Yaskawa INFORM job: A_ROOF_UPPER_0614_2_PL8.JBI

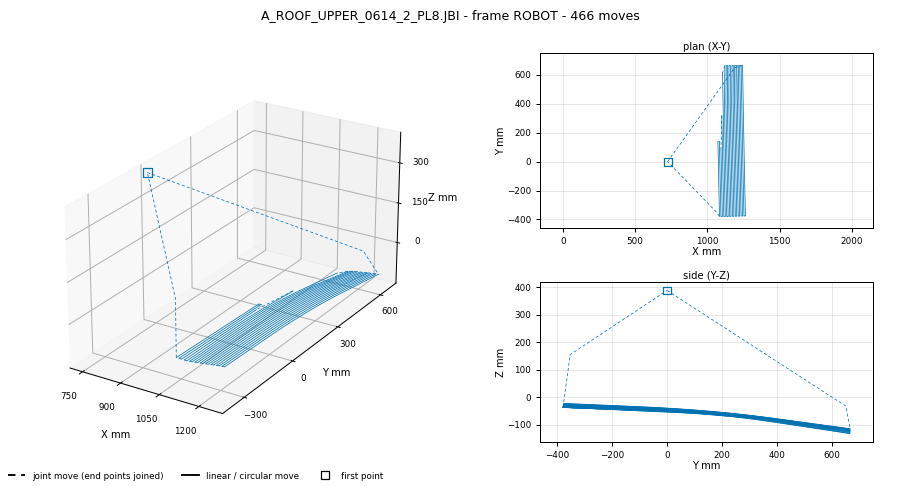
[picture p0: tool path of A_ROOF_UPPER_0614_2_PL8.JBI in frame ROBOT, 466 of 466 moves have a stored position in this frame; points joined in program order, loops and branches not executed]
/JOB
//NAME A_ROOF_UPPER_0614_2_PL8
//POS
///NPOS 466,0,0,0,0,0
///TOOL 0
///USER 0
///POSTYPE ROBOT
///RECTAN
///RCONF 1,0,0,0,0,0,0,0,0,0,0,0,0,0,0,0,0,0,0,0,0,0,0,0
C00000=725.000,0.000,388.500,-180.000,-0.000,0.000
///USER 0
///POSTYPE ROBOT
///RECTAN
C00001=1189.429,650.218,-32.227,172.053,-4.343,0.974
C00002=1243.739,665.281,-114.128,172.020,-4.282,1.414
C00003=1244.570,615.748,-107.360,172.042,-4.322,1.126
C00004=1248.336,391.180,-76.679,172.246,-4.167,0.979
C00005=1248.738,367.260,-73.517,172.471,-4.008,0.970
C00006=1249.092,346.433,-70.842,172.708,-3.888,0.966
C00007=1249.451,325.475,-68.240,172.968,-3.789,0.966
C00008=1249.796,305.508,-65.842,173.226,-3.716,0.968
C00009=1250.146,285.539,-63.530,173.487,-3.660,0.973
C00010=1250.497,265.663,-61.313,173.744,-3.621,0.979
C00011=1250.856,245.682,-59.173,174.000,-3.596,0.988
C00012=1251.235,224.702,-57.018,174.263,-3.583,0.998
C00013=1251.619,203.718,-54.952,174.521,-3.582,1.010
C00014=1252.006,182.729,-52.977,174.773,-3.593,1.023
C00015=1252.415,160.820,-51.011,175.027,-3.617,1.037
C00016=1252.831,138.821,-49.128,175.274,-3.653,1.053
C00017=1253.250,116.819,-47.334,175.514,-3.702,1.070
C00018=1253.692,93.813,-45.555,175.757,-3.765,1.088
C00019=1254.138,70.801,-43.865,175.991,-3.840,1.107
C00020=1254.589,47.783,-42.265,176.219,-3.924,1.127
C00021=1255.064,23.760,-40.691,176.449,-4.023,1.148
C00022=1255.542,-0.269,-39.207,176.673,-4.129,1.169
C00023=1256.026,-24.305,-37.813,176.890,-4.242,1.190
C00024=1256.533,-49.345,-36.455,177.109,-4.364,1.211
C00025=1257.044,-74.393,-35.191,177.323,-4.490,1.232
C00026=1257.558,-99.363,-34.023,177.531,-4.617,1.253
C00027=1262.246,-325.192,-24.300,177.735,-4.744,1.362
C00028=1263.282,-375.135,-22.149,177.733,-4.743,1.386
C00029=1253.337,-375.387,-23.203,177.732,-4.743,1.394
C00030=1252.299,-325.442,-25.310,177.735,-4.744,1.363
C00031=1247.595,-99.606,-34.838,177.531,-4.617,1.253
C00032=1247.079,-74.637,-35.984,177.323,-4.490,1.233
C00033=1246.565,-49.589,-37.227,177.109,-4.364,1.211
C00034=1246.057,-24.549,-38.563,176.890,-4.242,1.190
C00035=1245.572,-0.513,-39.937,176.673,-4.129,1.169
C00036=1245.092,23.516,-41.404,176.449,-4.023,1.148
C00037=1244.616,47.539,-42.961,176.219,-3.924,1.127
C00038=1244.165,70.557,-44.547,175.991,-3.840,1.107
C00039=1243.718,93.569,-46.224,175.757,-3.765,1.088
C00040=1243.275,116.575,-47.994,175.514,-3.702,1.070
C00041=1242.855,138.578,-49.780,175.274,-3.653,1.053
C00042=1242.439,160.575,-51.657,175.027,-3.617,1.037
C00043=1242.030,182.485,-53.620,174.773,-3.593,1.022
C00044=1241.642,203.473,-55.593,174.521,-3.582,1.009
C00045=1241.259,224.457,-57.659,174.263,-3.583,0.997
C00046=1240.879,245.434,-59.817,174.000,-3.596,0.986
C00047=1240.523,265.414,-61.962,173.744,-3.621,0.978
C00048=1240.171,285.288,-64.184,173.487,-3.660,0.971
C00049=1239.822,305.255,-66.507,173.226,-3.716,0.966
C00050=1239.477,325.219,-68.917,172.968,-3.789,0.964
C00051=1239.119,346.174,-71.538,172.709,-3.888,0.964
C00052=1238.768,366.999,-74.233,172.472,-4.008,0.968
C00053=1238.368,390.913,-77.423,172.246,-4.167,0.975
C00054=1234.646,615.465,-108.292,172.043,-4.324,1.109
C00055=1233.823,664.993,-115.099,172.011,-4.264,1.539
C00056=1223.907,664.704,-116.071,172.022,-4.285,1.389
C00057=1224.720,615.181,-109.222,172.045,-4.328,1.079
C00058=1228.400,390.647,-78.167,172.246,-4.168,0.972
C00059=1228.796,366.737,-74.949,172.472,-4.009,0.965
C00060=1229.147,345.916,-72.234,172.709,-3.889,0.962
C00061=1229.504,324.965,-69.594,172.968,-3.790,0.962
C00062=1229.847,305.004,-67.172,173.227,-3.716,0.964
C00063=1230.195,285.038,-64.840,173.487,-3.661,0.969
C00064=1230.546,265.166,-62.611,173.745,-3.622,0.976
C00065=1230.903,245.187,-60.461,174.000,-3.596,0.985
C00066=1231.282,224.210,-58.299,174.263,-3.583,0.996
C00067=1231.666,203.228,-56.234,174.521,-3.582,1.008
C00068=1232.054,182.240,-54.262,174.773,-3.593,1.021
C00069=1232.463,160.332,-52.302,175.027,-3.617,1.036
C00070=1232.880,138.334,-50.431,175.275,-3.653,1.052
C00071=1233.299,116.331,-48.654,175.514,-3.703,1.069
C00072=1233.743,93.326,-46.894,175.757,-3.765,1.088
C00073=1234.191,70.313,-45.228,175.991,-3.840,1.107
C00074=1234.644,47.295,-43.657,176.219,-3.924,1.127
C00075=1235.121,23.272,-42.115,176.449,-4.023,1.148
C00076=1235.601,-0.756,-40.668,176.673,-4.129,1.169
C00077=1236.087,-24.792,-39.313,176.890,-4.242,1.190
C00078=1236.598,-49.832,-37.998,177.109,-4.364,1.211
C00079=1237.113,-74.880,-36.777,177.323,-4.490,1.233
C00080=1237.630,-99.850,-35.654,177.531,-4.617,1.253
C00081=1242.351,-325.692,-26.320,177.734,-4.744,1.364
C00082=1243.394,-375.638,-24.255,177.733,-4.743,1.386
C00083=1233.450,-375.899,-25.309,177.782,-4.867,1.385
C00084=1232.404,-325.951,-27.330,177.783,-4.867,1.369
C00085=1227.667,-100.100,-36.468,177.580,-4.745,1.262
C00086=1227.148,-75.130,-37.570,177.372,-4.623,1.242
C00087=1226.631,-50.081,-38.769,177.158,-4.501,1.221
C00088=1226.118,-25.039,-40.063,176.937,-4.382,1.200
C00089=1225.631,-1.002,-41.397,176.718,-4.273,1.180
C00090=1225.149,23.028,-42.827,176.492,-4.172,1.159
C00091=1224.691,46.055,-44.287,176.267,-4.082,1.140
C00092=1224.236,69.074,-45.840,176.036,-4.001,1.121
C00093=1223.787,92.088,-47.487,175.796,-3.931,1.102
C00094=1223.362,114.097,-49.155,175.560,-3.875,1.085
C00095=1222.940,136.101,-50.915,175.316,-3.831,1.069
C00096=1222.525,158.020,-52.764,175.065,-3.798,1.053
C00097=1222.133,179.014,-54.627,174.817,-3.780,1.040
C00098=1221.744,200.003,-56.583,174.561,-3.772,1.027
C00099=1221.360,220.986,-58.635,174.297,-3.778,1.016
C00100=1220.997,240.970,-60.681,174.042,-3.795,1.006
C00101=1220.642,260.854,-62.807,173.783,-3.823,0.998
C00102=1220.289,280.824,-65.035,173.517,-3.865,0.991
C00103=1219.941,300.791,-67.357,173.248,-3.923,0.987
C00104=1219.596,320.754,-69.774,172.980,-3.998,0.984
C00105=1219.259,340.595,-72.269,172.721,-4.092,0.984
C00106=1218.907,361.536,-74.999,172.465,-4.215,0.988
C00107=1218.527,384.455,-78.089,172.229,-4.375,0.996
C00108=1217.998,417.090,-82.628,171.990,-4.603,1.009
C00109=1214.953,615.116,-110.490,171.985,-4.594,1.073
C00110=1214.190,664.623,-117.456,171.968,-4.565,1.281
C00111=1204.182,664.600,-118.494,171.912,-4.846,1.173
C00112=1204.954,615.099,-111.491,171.922,-4.863,1.056
C00113=1208.251,403.160,-81.508,172.008,-4.769,1.030
C00114=1208.674,377.272,-77.910,172.222,-4.570,1.018
C00115=1209.020,356.332,-75.085,172.461,-4.421,1.011
C00116=1209.355,336.382,-72.485,172.722,-4.302,1.007
C00117=1209.692,316.541,-69.991,172.994,-4.207,1.007
C00118=1210.019,297.569,-67.698,173.257,-4.134,1.009
C00119=1210.368,277.602,-65.380,173.534,-4.072,1.013
C00120=1210.721,257.629,-63.159,173.806,-4.026,1.019
C00121=1211.077,237.745,-61.042,174.070,-3.993,1.027
C00122=1211.440,217.760,-59.007,174.331,-3.972,1.035
C00123=1211.806,197.771,-57.062,174.586,-3.962,1.046
C00124=1212.195,176.781,-55.116,174.847,-3.965,1.057
C00125=1212.589,155.786,-53.265,175.100,-3.979,1.070
C00126=1212.985,134.863,-51.512,175.345,-4.006,1.084
C00127=1213.407,112.858,-49.764,175.594,-4.045,1.100
C00128=1213.834,90.847,-48.109,175.835,-4.097,1.116
C00129=1214.265,68.830,-46.548,176.068,-4.159,1.133
C00130=1214.720,45.809,-45.009,176.304,-4.235,1.152
C00131=1215.179,22.782,-43.565,176.532,-4.321,1.171
C00132=1215.663,-1.249,-42.153,176.761,-4.418,1.190
C00133=1216.152,-25.287,-40.836,176.983,-4.522,1.210
C00134=1216.665,-50.331,-39.564,177.205,-4.636,1.231
C00135=1217.184,-75.381,-38.386,177.421,-4.753,1.251
C00136=1217.705,-100.353,-37.305,177.628,-4.871,1.270
C00137=1222.459,-326.211,-28.354,177.830,-4.989,1.374
C00138=1223.509,-376.162,-26.375,177.829,-4.988,1.386
C00139=1213.569,-376.423,-27.454,177.874,-5.109,1.389
C00140=1212.515,-326.472,-29.394,177.875,-5.109,1.379
C00141=1207.745,-100.606,-38.163,177.674,-4.996,1.279
C00142=1207.223,-75.634,-39.224,177.467,-4.883,1.260
C00143=1206.702,-50.583,-40.382,177.251,-4.771,1.240
C00144=1206.187,-25.538,-41.635,177.027,-4.662,1.220
C00145=1205.697,-1.499,-42.934,176.803,-4.562,1.201
C00146=1205.211,22.535,-44.329,176.570,-4.469,1.182
C00147=1204.751,45.563,-45.759,176.339,-4.389,1.164
C00148=1204.295,68.585,-47.284,176.099,-4.318,1.146
C00149=1203.863,90.602,-48.835,175.861,-4.260,1.130
C00150=1203.436,112.614,-50.480,175.615,-4.214,1.114
C00151=1203.033,133.622,-52.140,175.372,-4.180,1.100
C00152=1202.635,154.546,-53.884,175.122,-4.159,1.087
C00153=1202.241,175.542,-55.729,174.864,-4.149,1.074
C00154=1201.870,195.536,-57.576,174.610,-4.151,1.064
C00155=1201.503,215.526,-59.512,174.349,-4.166,1.055
C00156=1201.143,235.421,-61.533,174.085,-4.191,1.046
C00157=1200.784,255.397,-63.656,173.813,-4.230,1.040
C00158=1200.449,274.376,-65.763,173.549,-4.279,1.035
C00159=1200.118,293.351,-67.959,173.279,-4.341,1.032
C00160=1199.793,312.213,-70.232,173.009,-4.416,1.030
C00161=1199.471,331.175,-72.609,172.739,-4.507,1.030
C00162=1199.153,350.136,-75.076,172.477,-4.618,1.033
C00163=1198.823,370.087,-77.763,172.221,-4.761,1.040
C00164=1198.434,393.997,-81.090,171.994,-4.957,1.052
C00165=1198.074,417.105,-84.377,171.858,-5.130,1.063
C00166=1198.550,615.125,-112.440,171.859,-5.131,1.053
C00167=1198.667,664.630,-119.456,171.852,-5.120,1.130
C00168=1189.050,664.613,-120.644,171.795,-5.403,1.029
C00169=1188.865,615.115,-113.579,171.795,-5.403,1.027
C00170=1188.115,416.320,-85.209,171.793,-5.389,1.090
C00171=1188.557,388.647,-81.242,171.950,-5.168,1.076
C00172=1188.910,366.863,-78.195,172.180,-4.979,1.064
C00173=1189.221,347.902,-75.628,172.441,-4.841,1.057
C00174=1189.538,328.941,-73.152,172.717,-4.729,1.054
C00175=1189.860,309.978,-70.769,172.996,-4.635,1.053
C00176=1190.184,291.118,-68.492,173.272,-4.556,1.054
C00177=1190.515,272.142,-66.294,173.548,-4.489,1.056
C00178=1190.851,253.162,-64.188,173.818,-4.433,1.060
C00179=1191.209,233.186,-62.068,174.096,-4.389,1.066
C00180=1191.569,213.291,-60.053,174.367,-4.359,1.074
C00181=1191.936,193.300,-58.122,174.632,-4.340,1.082
C00182=1192.308,173.305,-56.284,174.891,-4.334,1.092
C00183=1192.703,152.308,-54.451,175.154,-4.339,1.104
C00184=1193.103,131.306,-52.712,175.410,-4.356,1.116
C00185=1193.505,110.373,-51.073,175.656,-4.386,1.130
C00186=1193.933,88.361,-49.445,175.906,-4.429,1.145
C00187=1194.366,66.342,-47.912,176.149,-4.482,1.160
C00188=1194.804,44.317,-46.471,176.382,-4.546,1.177
C00189=1195.266,21.288,-45.059,176.617,-4.622,1.194
C00190=1195.732,-1.749,-43.739,176.843,-4.707,1.212
C00191=1196.224,-25.789,-42.458,177.069,-4.801,1.230
C00192=1196.720,-49.837,-41.271,177.286,-4.902,1.249
C00193=1197.240,-74.806,-40.133,177.502,-5.009,1.268
C00194=1197.787,-100.862,-39.044,177.719,-5.121,1.287
C00195=1202.573,-326.734,-30.447,177.917,-5.229,1.384
C00196=1203.630,-376.687,-28.546,177.916,-5.228,1.394
C00197=1193.692,-376.950,-29.649,177.957,-5.346,1.400
C00198=1192.632,-326.997,-31.513,177.958,-5.347,1.390
C00199=1187.832,-101.118,-39.946,177.760,-5.245,1.295
C00200=1187.282,-75.061,-41.016,177.544,-5.138,1.276
C00201=1186.761,-50.091,-42.135,177.328,-5.036,1.258
C00202=1186.263,-26.043,-43.305,177.109,-4.941,1.240
C00203=1185.770,-2.000,-44.570,176.880,-4.851,1.222
C00204=1185.302,21.036,-45.876,176.651,-4.772,1.205
C00205=1184.839,44.067,-47.274,176.412,-4.701,1.189
C00206=1184.401,66.092,-48.705,176.175,-4.641,1.173
C00207=1183.967,88.111,-50.228,175.928,-4.593,1.158
C00208=1183.558,109.128,-51.774,175.684,-4.556,1.144
C00209=1183.154,130.061,-53.404,175.433,-4.531,1.132
C00210=1182.755,151.064,-55.134,175.172,-4.518,1.120
C00211=1182.378,171.066,-56.872,174.916,-4.517,1.110
C00212=1182.005,191.061,-58.703,174.652,-4.528,1.100
C00213=1181.638,211.053,-60.627,174.382,-4.551,1.092
C00214=1181.277,230.948,-62.638,174.105,-4.587,1.086
C00215=1180.937,249.931,-64.649,173.835,-4.633,1.081
C00216=1180.602,268.912,-66.750,173.559,-4.693,1.078
C00217=1180.273,287.783,-68.933,173.280,-4.765,1.076
C00218=1179.947,306.749,-71.221,172.995,-4.849,1.076
C00219=1179.626,325.713,-73.605,172.709,-4.946,1.077
C00220=1179.310,344.675,-76.086,172.422,-5.059,1.081
C00221=1179.002,363.500,-78.644,172.142,-5.195,1.087
C00222=1178.681,383.439,-81.448,171.901,-5.376,1.099
C00223=1178.163,416.202,-86.182,171.725,-5.655,1.118
C00224=1179.134,615.111,-114.770,171.734,-5.679,1.000
C00225=1179.376,664.602,-121.883,171.741,-5.689,0.926
C00226=1170.628,664.605,-123.074,171.686,-5.975,0.835
C00227=1170.148,615.119,-115.932,171.671,-5.954,0.981
C00228=1168.215,416.580,-87.274,171.655,-5.926,1.146
C00229=1168.414,403.116,-85.300,171.691,-5.823,1.140
C00230=1168.838,376.249,-81.401,171.878,-5.557,1.120
C00231=1169.127,358.289,-78.872,172.140,-5.399,1.110
C00232=1169.418,340.455,-76.449,172.419,-5.274,1.104
C00233=1169.717,322.482,-74.096,172.700,-5.164,1.101
C00234=1170.020,304.510,-71.832,172.979,-5.068,1.099
C00235=1170.346,285.544,-69.539,173.269,-4.978,1.098
C00236=1170.674,266.673,-67.354,173.554,-4.901,1.099
C00237=1171.009,247.692,-65.252,173.836,-4.835,1.101
C00238=1171.348,228.709,-63.243,174.112,-4.784,1.106
C00239=1171.693,209.721,-61.325,174.381,-4.745,1.111
C00240=1172.059,189.817,-59.410,174.657,-4.717,1.118
C00241=1172.431,169.819,-57.583,174.926,-4.701,1.127
C00242=1172.808,149.818,-55.849,175.188,-4.697,1.136
C00243=1173.189,129.811,-54.204,175.442,-4.705,1.147
C00244=1173.593,108.878,-52.579,175.698,-4.725,1.159
C00245=1174.003,87.862,-51.040,175.948,-4.757,1.172
C00246=1174.437,65.841,-49.525,176.199,-4.801,1.186
C00247=1174.876,43.815,-48.104,176.441,-4.855,1.201
C00248=1175.340,20.784,-46.718,176.683,-4.921,1.217
C00249=1175.810,-2.254,-45.427,176.915,-4.996,1.233
C00250=1176.304,-26.298,-44.177,177.146,-5.081,1.250
C00251=1176.803,-50.347,-43.023,177.367,-5.171,1.267
C00252=1177.327,-75.317,-41.921,177.585,-5.267,1.285
C00253=1177.877,-101.376,-40.869,177.800,-5.367,1.302
C00254=1182.692,-327.261,-32.593,177.997,-5.464,1.395
C00255=1183.756,-377.215,-30.762,177.996,-5.464,1.407
C00256=1173.821,-377.482,-31.885,178.031,-5.581,1.415
C00257=1172.755,-327.525,-33.683,178.033,-5.581,1.401
C00258=1167.926,-101.635,-41.814,177.838,-5.490,1.310
C00259=1167.372,-75.576,-42.848,177.622,-5.395,1.293
C00260=1166.847,-50.605,-43.934,177.404,-5.305,1.276
C00261=1166.347,-26.554,-45.073,177.182,-5.221,1.260
C00262=1165.871,-3.508,-46.255,176.958,-5.145,1.244
C00263=1165.401,19.531,-47.529,176.724,-5.075,1.229
C00264=1164.956,41.565,-48.839,176.489,-5.015,1.214
C00265=1164.515,63.594,-50.241,176.243,-4.965,1.200
C00266=1164.099,84.617,-51.669,176.000,-4.926,1.187
C00267=1163.690,105.558,-53.184,175.747,-4.897,1.175
C00268=1163.284,126.569,-54.798,175.485,-4.880,1.163
C00269=1162.902,146.577,-56.427,175.228,-4.875,1.153
C00270=1162.524,166.580,-58.148,174.961,-4.882,1.144
C00271=1162.152,186.577,-59.964,174.687,-4.902,1.136
C00272=1161.803,205.488,-61.772,174.421,-4.932,1.130
C00273=1161.459,224.477,-63.678,174.146,-4.975,1.126
C00274=1161.119,243.462,-65.675,173.865,-5.030,1.122
C00275=1160.784,262.444,-67.770,173.576,-5.099,1.120
C00276=1160.455,281.316,-69.947,173.286,-5.180,1.120
C00277=1160.147,299.292,-72.114,173.005,-5.269,1.121
C00278=1159.843,317.267,-74.370,172.722,-5.369,1.124
C00279=1159.547,335.113,-76.700,172.436,-5.482,1.128
C00280=1159.254,353.076,-79.137,172.145,-5.609,1.134
C00281=1158.982,370.049,-81.526,171.867,-5.747,1.142
C00282=1158.672,389.838,-84.407,171.642,-5.956,1.158
C00283=1158.272,415.709,-88.232,171.585,-6.187,1.174
C00284=1159.271,615.118,-117.349,171.606,-6.230,0.958
C00285=1159.517,664.594,-124.574,171.633,-6.267,0.706
C00286=1149.612,664.593,-126.030,171.572,-6.554,0.588
C00287=1149.358,615.127,-118.743,171.531,-6.500,0.952
C00288=1148.334,415.437,-89.323,171.506,-6.448,1.202
C00289=1148.805,384.623,-84.721,171.566,-6.150,1.180
C00290=1149.083,366.815,-82.112,171.830,-5.974,1.167
C00291=1149.353,349.841,-79.714,172.120,-5.836,1.159
C00292=1149.644,331.877,-77.270,172.418,-5.703,1.152
C00293=1149.941,314.032,-74.935,172.710,-5.583,1.147
C00294=1150.243,296.056,-72.677,173.000,-5.477,1.143
C00295=1150.550,278.079,-70.510,173.287,-5.384,1.141
C00296=1150.862,260.101,-68.434,173.570,-5.303,1.141
C00297=1151.195,241.218,-66.349,173.862,-5.230,1.142
C00298=1151.535,222.233,-64.351,174.150,-5.170,1.145
C00299=1151.880,203.243,-62.447,174.430,-5.122,1.149
C00300=1152.228,184.332,-60.644,174.702,-5.087,1.154
C00301=1152.582,165.330,-58.922,174.969,-5.064,1.161
C00302=1152.960,145.327,-57.205,175.240,-5.053,1.169
C00303=1153.342,125.319,-55.581,175.504,-5.054,1.178
C00304=1153.730,105.304,-54.049,175.758,-5.066,1.189
C00305=1154.140,84.363,-52.539,176.015,-5.090,1.200
C00306=1154.557,63.338,-51.116,176.264,-5.125,1.213
C00307=1154.998,41.310,-49.724,176.513,-5.170,1.226
C00308=1155.444,19.275,-48.424,176.751,-5.225,1.240
C00309=1155.915,-3.765,-47.162,176.989,-5.290,1.255
C00310=1156.392,-26.812,-45.994,177.215,-5.361,1.270
C00311=1156.895,-50.864,-44.869,177.439,-5.439,1.285
C00312=1157.421,-75.835,-43.798,177.658,-5.524,1.301
C00313=1157.975,-101.896,-42.781,177.872,-5.612,1.318
C00314=1162.819,-327.791,-34.786,178.067,-5.697,1.406
C00315=1163.889,-377.749,-33.019,178.065,-5.696,1.424
C00316=1153.956,-378.015,-34.144,178.095,-5.810,1.435
C00317=1152.884,-328.057,-35.887,178.098,-5.811,1.410
C00318=1148.006,-101.159,-43.805,177.897,-5.731,1.324
C00319=1147.450,-75.098,-44.811,177.682,-5.649,1.309
C00320=1146.921,-50.041,-45.875,177.461,-5.570,1.294
C00321=1146.419,-26.072,-46.986,177.237,-5.497,1.279
C00322=1145.942,-3.026,-48.147,177.008,-5.432,1.265
C00323=1145.469,20.015,-49.402,176.766,-5.373,1.251
C00324=1145.022,42.051,-50.697,176.524,-5.324,1.237
C00325=1144.600,63.082,-52.021,176.282,-5.284,1.225
C00326=1144.183,84.106,-53.437,176.029,-5.255,1.214
C00327=1143.772,105.048,-54.942,175.767,-5.235,1.203
C00328=1143.384,125.062,-56.474,175.507,-5.228,1.193
C00329=1143.002,145.072,-58.097,175.237,-5.231,1.185
C00330=1142.643,164.078,-59.729,174.973,-5.247,1.178
C00331=1142.291,182.997,-61.442,174.702,-5.274,1.172
C00332=1141.941,201.991,-63.254,174.423,-5.314,1.167
C00333=1141.597,220.981,-65.161,174.135,-5.367,1.164
C00334=1141.275,238.973,-67.058,173.857,-5.429,1.162
C00335=1140.961,256.861,-69.032,173.575,-5.502,1.162
C00336=1140.649,274.841,-71.107,173.287,-5.586,1.163
C00337=1140.342,292.818,-73.275,172.993,-5.683,1.165
C00338=1140.042,310.675,-75.522,172.698,-5.793,1.169
C00339=1139.746,328.640,-77.877,172.397,-5.918,1.175
C00340=1139.471,345.614,-80.191,172.109,-6.051,1.183
C00341=1139.204,362.445,-82.572,171.817,-6.197,1.192
C00342=1138.941,379.408,-85.062,171.524,-6.352,1.203
C00343=1138.535,406.032,-89.076,171.344,-8.117,1.401
C00344=1138.400,415.917,-90.582,171.339,-8.283,1.418
C00345=1140.286,615.128,-120.237,171.373,-8.347,1.185
C00346=1140.753,664.582,-127.599,171.441,-8.417,0.720
C00347=1130.859,664.438,-129.965,171.213,-8.393,0.854
C00348=1130.391,615.012,-122.427,171.167,-8.345,1.167
C00349=1128.495,415.610,-92.013,171.142,-8.273,1.414
C00350=1128.845,391.183,-88.242,171.323,-7.974,1.385
C00351=1129.105,373.942,-85.634,171.528,-7.922,1.384
C00352=1129.376,356.411,-83.063,171.815,-7.904,1.386
C00353=1129.653,338.867,-80.585,172.115,-7.878,1.388
C00354=1129.947,320.597,-78.099,172.413,-7.846,1.388
C00355=1130.252,302.036,-75.673,172.713,-7.808,1.389
C00356=1130.562,283.463,-73.344,173.011,-7.768,1.388
C00357=1130.874,265.152,-71.147,173.304,-7.719,1.387
C00358=1131.196,246.555,-69.011,173.627,-7.662,1.385
C00359=1131.523,227.947,-66.969,173.903,-7.594,1.382
C00360=1131.869,208.607,-64.955,174.185,-7.493,1.377
C00361=1132.170,191.968,-63.300,174.454,-7.420,1.373
C00362=1132.512,173.331,-61.532,174.728,-7.324,1.368
C00363=1132.862,154.589,-59.848,175.016,-7.210,1.362
C00364=1133.257,133.814,-58.115,175.384,-5.404,1.205
C00365=1133.643,113.801,-56.544,175.655,-5.402,1.213
C00366=1134.042,93.323,-55.032,175.921,-5.412,1.222
C00367=1134.248,82.850,-54.296,176.052,-5.420,1.228
C00368=1134.666,61.825,-52.889,176.309,-5.446,1.239
C00369=1135.089,40.793,-51.575,176.555,-5.481,1.250
C00370=1135.536,18.757,-50.293,176.801,-5.525,1.262
C00371=1135.990,-3.285,-49.104,177.034,-5.577,1.275
C00372=1136.469,-26.333,-47.954,177.265,-5.637,1.289
C00373=1136.972,-50.303,-46.855,177.491,-5.704,1.303
C00374=1137.502,-75.360,-45.806,177.713,-5.776,1.317
C00375=1138.059,-101.422,-44.812,177.927,-5.852,1.332
C00376=1142.950,-328.325,-37.013,178.126,-5.926,1.414
C00377=1144.025,-378.284,-35.295,178.124,-5.926,1.433
C00378=1134.095,-378.553,-36.456,178.150,-6.040,1.432
C00379=1133.018,-328.593,-38.149,178.152,-6.040,1.418
C00380=1128.115,-101.686,-45.842,177.954,-5.973,1.339
C00381=1127.556,-75.574,-46.823,177.830,-4.400,1.222
C00382=1127.123,-55.297,-47.638,177.588,-4.743,1.236
C00383=1126.707,-35.594,-48.505,177.359,-5.057,1.250
C00384=1126.239,-13.173,-49.585,177.121,-5.392,1.265
C00385=1125.797,8.243,-50.711,176.879,-5.700,1.280
C00386=1125.396,27.932,-51.829,176.632,-5.969,1.293
C00387=1125.000,47.615,-53.031,176.381,-6.207,1.306
C00388=1124.594,68.013,-54.370,176.119,-6.433,1.318
C00389=1124.188,88.681,-55.821,175.864,-6.653,1.330
C00390=1123.812,108.068,-57.270,175.585,-6.839,1.340
C00391=1123.435,127.723,-58.838,175.314,-6.996,1.349
C00392=1123.050,148.089,-60.555,175.049,-7.159,1.359
C00393=1122.703,166.733,-62.219,174.762,-7.283,1.365
C00394=1122.347,186.083,-64.041,174.481,-7.389,1.371
C00395=1122.010,204.709,-65.886,174.200,-7.477,1.375
C00396=1121.678,223.325,-67.823,173.932,-7.569,1.380
C00397=1121.373,240.656,-69.712,173.650,-7.637,1.383
C00398=1121.062,258.691,-71.764,173.384,-7.699,1.385
C00399=1120.753,276.844,-73.918,173.095,-7.752,1.387
C00400=1120.446,295.136,-76.185,172.799,-7.793,1.387
C00401=1120.141,313.696,-78.581,172.502,-7.831,1.387
C00402=1119.840,332.242,-81.075,172.202,-7.866,1.386
C00403=1119.552,350.495,-83.626,171.904,-7.897,1.385
C00404=1119.281,368.026,-86.170,171.606,-7.915,1.383
C00405=1119.016,385.542,-88.803,171.332,-7.947,1.381
C00406=1118.801,400.084,-91.046,171.151,-8.043,1.388
C00407=1118.619,412.643,-93.022,170.986,-8.214,1.405
C00408=1118.593,415.606,-93.491,170.946,-8.268,1.410
C00409=1120.778,614.897,-124.574,170.959,-8.342,1.162
C00410=1121.318,664.296,-132.280,170.991,-8.376,0.944
C00411=1105.570,614.010,-123.215,171.652,-7.951,1.120
C00412=1106.334,564.532,-116.047,171.635,-7.933,1.243
C00413=1109.667,348.539,-84.757,171.918,-7.893,1.384
C00414=1109.959,330.009,-82.171,172.217,-7.862,1.385
C00415=1110.258,311.466,-79.683,172.515,-7.826,1.386
C00416=1110.558,293.195,-77.327,172.806,-7.788,1.386
C00417=1110.869,274.627,-75.028,173.100,-7.744,1.385
C00418=1111.184,256.046,-72.825,173.386,-7.688,1.384
C00419=1111.501,237.740,-70.744,173.655,-7.626,1.382
C00420=1111.809,220.132,-68.825,173.923,-7.549,1.378
C00421=1112.123,202.516,-66.989,174.194,-7.467,1.374
C00422=1112.471,183.184,-65.070,174.471,-7.373,1.369
C00423=1112.831,163.560,-63.216,174.744,-7.262,1.364
C00424=1113.172,145.205,-61.569,175.010,-7.132,1.356
C00425=1113.560,124.566,-59.813,175.275,-6.967,1.347
C00426=1113.915,105.914,-58.310,175.527,-6.816,1.338
C00427=1114.289,86.537,-56.838,175.783,-6.625,1.327
C00428=1114.693,65.877,-55.358,176.035,-6.405,1.315
C00429=1115.096,45.490,-53.989,176.289,-6.176,1.303
C00430=1115.509,24.816,-52.692,176.538,-5.921,1.290
C00431=1115.942,3.417,-51.441,176.785,-5.622,1.275
C00432=1116.365,-17.269,-50.320,177.021,-5.324,1.261
C00433=1116.829,-39.679,-49.199,177.262,-4.988,1.246
C00434=1117.318,-63.093,-48.127,177.504,-4.605,1.229
C00435=1117.778,-84.792,-47.225,177.742,-4.223,1.214
C00436=1118.299,-109.216,-46.306,177.963,-3.788,1.198
C00437=1123.026,-328.488,-38.851,178.153,-3.420,1.301
C00438=1124.102,-378.447,-37.152,178.152,-3.419,1.324
C00439=1114.039,-378.200,-37.108,177.952,-3.411,1.315
C00440=1112.977,-328.245,-38.938,177.953,-3.412,1.297
C00441=1108.496,-117.713,-46.648,177.858,-3.621,1.191
C00442=1108.001,-94.298,-47.571,177.645,-4.042,1.206
C00443=1107.511,-70.887,-48.581,177.420,-4.461,1.222
C00444=1107.040,-48.199,-49.653,177.190,-4.840,1.238
C00445=1106.600,-26.797,-50.745,176.973,-5.170,1.253
C00446=1106.160,-5.118,-51.939,176.736,-5.491,1.267
C00447=1105.729,16.272,-53.205,176.497,-5.798,1.283
C00448=1105.304,37.655,-54.560,176.261,-6.076,1.297
C00449=1104.898,58.318,-55.956,176.017,-6.316,1.310
C00450=1104.501,78.690,-57.421,175.764,-6.536,1.322
C00451=1104.105,99.339,-58.995,175.519,-6.750,1.334
C00452=1099.944,318.457,-76.674,175.270,-6.926,1.284
C00453=1094.176,89.157,-55.681,177.767,-3.412,1.051
C00454=1102.917,-327.991,-38.766,177.753,-3.402,1.292
C00455=1103.962,-377.939,-36.741,177.752,-3.402,1.308
C00456=1093.939,-378.145,-36.643,177.752,-3.402,1.301
C00457=1092.902,-328.203,-38.807,177.753,-3.403,1.287
C00458=1084.234,88.899,-56.878,177.616,-3.744,1.079
C00459=1083.195,138.841,-59.042,177.617,-3.745,1.050
C00460=1073.262,138.575,-60.377,177.617,-3.745,1.049
C00461=1074.292,88.639,-58.075,177.616,-3.744,1.078
C00462=1082.888,-328.413,-38.847,177.753,-3.403,1.282
C00463=1083.916,-378.349,-36.545,177.752,-3.402,1.294
C00464=1066.114,-352.262,155.451,177.759,-3.407,1.176
///USER 0
///POSTYPE ROBOT
///RECTAN
C00465=725.000,0.000,388.500,-180.000,-0.000,0.000
//INST
///DATE 2021/06/15 16:23
///ATTR SC,RW,RJ
////FRAME ROBOT
///GROUP1 RB1
NOP
MOVJ C00000 VJ=100.00 PL=0
'Path Start: Op_ID_1
MOVJ C00001 VJ=25.00 PL=0
MOVJ C00002 VJ=25.00 PL=0
MOVL C00003 V=800.0 PL=8
SPYON
MOVL C00004 V=800.0 PL=8
MOVL C00005 V=800.0 PL=8
MOVL C00006 V=800.0 PL=8
MOVL C00007 V=800.0 PL=8
MOVL C00008 V=800.0 PL=8
MOVL C00009 V=800.0 PL=8
MOVL C00010 V=800.0 PL=8
MOVL C00011 V=800.0 PL=8
MOVL C00012 V=800.0 PL=8
MOVL C00013 V=800.0 PL=8
MOVL C00014 V=800.0 PL=8
MOVL C00015 V=800.0 PL=8
MOVL C00016 V=800.0 PL=8
MOVL C00017 V=800.0 PL=8
MOVL C00018 V=800.0 PL=8
MOVL C00019 V=800.0 PL=8
MOVL C00020 V=800.0 PL=8
MOVL C00021 V=800.0 PL=8
MOVL C00022 V=800.0 PL=8
MOVL C00023 V=800.0 PL=8
MOVL C00024 V=800.0 PL=8
MOVL C00025 V=800.0 PL=8
MOVL C00026 V=800.0 PL=8
MOVL C00027 V=800.0 PL=8
SPYOF
MOVL C00028 V=800.0 PL=0
MOVJ C00029 VJ=25.00 PL=0
MOVL C00030 V=800.0 PL=8
SPYON
MOVL C00031 V=800.0 PL=8
MOVL C00032 V=800.0 PL=8
MOVL C00033 V=800.0 PL=8
MOVL C00034 V=800.0 PL=8
MOVL C00035 V=800.0 PL=8
MOVL C00036 V=800.0 PL=8
MOVL C00037 V=800.0 PL=8
MOVL C00038 V=800.0 PL=8
MOVL C00039 V=800.0 PL=8
MOVL C00040 V=800.0 PL=8
MOVL C00041 V=800.0 PL=8
MOVL C00042 V=800.0 PL=8
MOVL C00043 V=800.0 PL=8
MOVL C00044 V=800.0 PL=8
MOVL C00045 V=800.0 PL=8
MOVL C00046 V=800.0 PL=8
MOVL C00047 V=800.0 PL=8
MOVL C00048 V=800.0 PL=8
MOVL C00049 V=800.0 PL=8
MOVL C00050 V=800.0 PL=8
MOVL C00051 V=800.0 PL=8
MOVL C00052 V=800.0 PL=8
MOVL C00053 V=800.0 PL=8
MOVL C00054 V=800.0 PL=8
SPYOF
MOVL C00055 V=800.0 PL=0
MOVJ C00056 VJ=25.00 PL=0
MOVL C00057 V=800.0 PL=8
SPYON
MOVL C00058 V=800.0 PL=8
MOVL C00059 V=800.0 PL=8
MOVL C00060 V=800.0 PL=8
MOVL C00061 V=800.0 PL=8
MOVL C00062 V=800.0 PL=8
MOVL C00063 V=800.0 PL=8
MOVL C00064 V=800.0 PL=8
MOVL C00065 V=800.0 PL=8
MOVL C00066 V=800.0 PL=8
MOVL C00067 V=800.0 PL=8
MOVL C00068 V=800.0 PL=8
MOVL C00069 V=800.0 PL=8
MOVL C00070 V=800.0 PL=8
MOVL C00071 V=800.0 PL=8
MOVL C00072 V=800.0 PL=8
MOVL C00073 V=800.0 PL=8
MOVL C00074 V=800.0 PL=8
MOVL C00075 V=800.0 PL=8
MOVL C00076 V=800.0 PL=8
MOVL C00077 V=800.0 PL=8
MOVL C00078 V=800.0 PL=8
MOVL C00079 V=800.0 PL=8
MOVL C00080 V=800.0 PL=8
MOVL C00081 V=800.0 PL=8
SPYOF
MOVL C00082 V=800.0 PL=0
MOVJ C00083 VJ=25.00 PL=0
MOVL C00084 V=800.0 PL=8
SPYON
MOVL C00085 V=800.0 PL=8
MOVL C00086 V=800.0 PL=8
MOVL C00087 V=800.0 PL=8
MOVL C00088 V=800.0 PL=8
MOVL C00089 V=800.0 PL=8
MOVL C00090 V=800.0 PL=8
MOVL C00091 V=800.0 PL=8
MOVL C00092 V=800.0 PL=8
MOVL C00093 V=800.0 PL=8
MOVL C00094 V=800.0 PL=8
MOVL C00095 V=800.0 PL=8
MOVL C00096 V=800.0 PL=8
MOVL C00097 V=800.0 PL=8
MOVL C00098 V=800.0 PL=8
MOVL C00099 V=800.0 PL=8
MOVL C00100 V=800.0 PL=8
MOVL C00101 V=800.0 PL=8
MOVL C00102 V=800.0 PL=8
MOVL C00103 V=800.0 PL=8
MOVL C00104 V=800.0 PL=8
MOVL C00105 V=800.0 PL=8
MOVL C00106 V=800.0 PL=8
MOVL C00107 V=800.0 PL=8
MOVL C00108 V=800.0 PL=8
MOVL C00109 V=800.0 PL=8
SPYOF
MOVL C00110 V=800.0 PL=0
MOVJ C00111 VJ=25.00 PL=0
MOVL C00112 V=800.0 PL=8
SPYON
MOVL C00113 V=800.0 PL=8
MOVL C00114 V=800.0 PL=8
MOVL C00115 V=800.0 PL=8
MOVL C00116 V=800.0 PL=8
MOVL C00117 V=800.0 PL=8
MOVL C00118 V=800.0 PL=8
MOVL C00119 V=800.0 PL=8
MOVL C00120 V=800.0 PL=8
MOVL C00121 V=800.0 PL=8
MOVL C00122 V=800.0 PL=8
MOVL C00123 V=800.0 PL=8
MOVL C00124 V=800.0 PL=8
MOVL C00125 V=800.0 PL=8
MOVL C00126 V=800.0 PL=8
MOVL C00127 V=800.0 PL=8
MOVL C00128 V=800.0 PL=8
MOVL C00129 V=800.0 PL=8
MOVL C00130 V=800.0 PL=8
MOVL C00131 V=800.0 PL=8
MOVL C00132 V=800.0 PL=8
MOVL C00133 V=800.0 PL=8
MOVL C00134 V=800.0 PL=8
MOVL C00135 V=800.0 PL=8
MOVL C00136 V=800.0 PL=8
MOVL C00137 V=800.0 PL=8
SPYOF
MOVL C00138 V=800.0 PL=0
MOVJ C00139 VJ=25.00 PL=0
MOVL C00140 V=800.0 PL=8
SPYON
MOVL C00141 V=800.0 PL=8
MOVL C00142 V=800.0 PL=8
MOVL C00143 V=800.0 PL=8
MOVL C00144 V=800.0 PL=8
MOVL C00145 V=800.0 PL=8
MOVL C00146 V=800.0 PL=8
MOVL C00147 V=800.0 PL=8
MOVL C00148 V=800.0 PL=8
MOVL C00149 V=800.0 PL=8
MOVL C00150 V=800.0 PL=8
MOVL C00151 V=800.0 PL=8
MOVL C00152 V=800.0 PL=8
MOVL C00153 V=800.0 PL=8
MOVL C00154 V=800.0 PL=8
MOVL C00155 V=800.0 PL=8
MOVL C00156 V=800.0 PL=8
MOVL C00157 V=800.0 PL=8
MOVL C00158 V=800.0 PL=8
MOVL C00159 V=800.0 PL=8
MOVL C00160 V=800.0 PL=8
MOVL C00161 V=800.0 PL=8
MOVL C00162 V=800.0 PL=8
MOVL C00163 V=800.0 PL=8
MOVL C00164 V=800.0 PL=8
MOVL C00165 V=800.0 PL=8
MOVL C00166 V=800.0 PL=8
SPYOF
MOVL C00167 V=800.0 PL=0
MOVJ C00168 VJ=25.00 PL=0
MOVL C00169 V=800.0 PL=8
SPYON
MOVL C00170 V=800.0 PL=8
MOVL C00171 V=800.0 PL=8
MOVL C00172 V=800.0 PL=8
MOVL C00173 V=800.0 PL=8
MOVL C00174 V=800.0 PL=8
MOVL C00175 V=800.0 PL=8
MOVL C00176 V=800.0 PL=8
MOVL C00177 V=800.0 PL=8
MOVL C00178 V=800.0 PL=8
MOVL C00179 V=800.0 PL=8
MOVL C00180 V=800.0 PL=8
MOVL C00181 V=800.0 PL=8
MOVL C00182 V=800.0 PL=8
MOVL C00183 V=800.0 PL=8
MOVL C00184 V=800.0 PL=8
MOVL C00185 V=800.0 PL=8
MOVL C00186 V=800.0 PL=8
MOVL C00187 V=800.0 PL=8
MOVL C00188 V=800.0 PL=8
MOVL C00189 V=800.0 PL=8
MOVL C00190 V=800.0 PL=8
MOVL C00191 V=800.0 PL=8
MOVL C00192 V=800.0 PL=8
MOVL C00193 V=800.0 PL=8
MOVL C00194 V=800.0 PL=8
MOVL C00195 V=800.0 PL=8
SPYOF
MOVL C00196 V=800.0 PL=0
MOVJ C00197 VJ=25.00 PL=0
MOVL C00198 V=800.0 PL=8
SPYON
MOVL C00199 V=800.0 PL=8
MOVL C00200 V=800.0 PL=8
MOVL C00201 V=800.0 PL=8
MOVL C00202 V=800.0 PL=8
MOVL C00203 V=800.0 PL=8
MOVL C00204 V=800.0 PL=8
MOVL C00205 V=800.0 PL=8
MOVL C00206 V=800.0 PL=8
MOVL C00207 V=800.0 PL=8
MOVL C00208 V=800.0 PL=8
MOVL C00209 V=800.0 PL=8
MOVL C00210 V=800.0 PL=8
MOVL C00211 V=800.0 PL=8
MOVL C00212 V=800.0 PL=8
MOVL C00213 V=800.0 PL=8
MOVL C00214 V=800.0 PL=8
MOVL C00215 V=800.0 PL=8
MOVL C00216 V=800.0 PL=8
MOVL C00217 V=800.0 PL=8
MOVL C00218 V=800.0 PL=8
MOVL C00219 V=800.0 PL=8
MOVL C00220 V=800.0 PL=8
MOVL C00221 V=800.0 PL=8
MOVL C00222 V=800.0 PL=8
MOVL C00223 V=800.0 PL=8
MOVL C00224 V=800.0 PL=8
SPYOF
MOVL C00225 V=800.0 PL=0
MOVJ C00226 VJ=25.00 PL=0
MOVL C00227 V=800.0 PL=8
SPYON
MOVL C00228 V=800.0 PL=8
MOVL C00229 V=800.0 PL=8
MOVL C00230 V=800.0 PL=8
MOVL C00231 V=800.0 PL=8
MOVL C00232 V=800.0 PL=8
MOVL C00233 V=800.0 PL=8
MOVL C00234 V=800.0 PL=8
MOVL C00235 V=800.0 PL=8
MOVL C00236 V=800.0 PL=8
MOVL C00237 V=800.0 PL=8
MOVL C00238 V=800.0 PL=8
MOVL C00239 V=800.0 PL=8
MOVL C00240 V=800.0 PL=8
MOVL C00241 V=800.0 PL=8
MOVL C00242 V=800.0 PL=8
MOVL C00243 V=800.0 PL=8
MOVL C00244 V=800.0 PL=8
MOVL C00245 V=800.0 PL=8
MOVL C00246 V=800.0 PL=8
MOVL C00247 V=800.0 PL=8
MOVL C00248 V=800.0 PL=8
MOVL C00249 V=800.0 PL=8
MOVL C00250 V=800.0 PL=8
MOVL C00251 V=800.0 PL=8
MOVL C00252 V=800.0 PL=8
MOVL C00253 V=800.0 PL=8
MOVL C00254 V=800.0 PL=8
SPYOF
MOVL C00255 V=800.0 PL=0
MOVJ C00256 VJ=25.00 PL=0
MOVL C00257 V=800.0 PL=8
SPYON
MOVL C00258 V=800.0 PL=8
MOVL C00259 V=800.0 PL=8
MOVL C00260 V=800.0 PL=8
MOVL C00261 V=800.0 PL=8
MOVL C00262 V=800.0 PL=8
MOVL C00263 V=800.0 PL=8
MOVL C00264 V=800.0 PL=8
MOVL C00265 V=800.0 PL=8
MOVL C00266 V=800.0 PL=8
MOVL C00267 V=800.0 PL=8
MOVL C00268 V=800.0 PL=8
MOVL C00269 V=800.0 PL=8
MOVL C00270 V=800.0 PL=8
MOVL C00271 V=800.0 PL=8
MOVL C00272 V=800.0 PL=8
MOVL C00273 V=800.0 PL=8
MOVL C00274 V=800.0 PL=8
MOVL C00275 V=800.0 PL=8
MOVL C00276 V=800.0 PL=8
MOVL C00277 V=800.0 PL=8
MOVL C00278 V=800.0 PL=8
MOVL C00279 V=800.0 PL=8
MOVL C00280 V=800.0 PL=8
MOVL C00281 V=800.0 PL=8
MOVL C00282 V=800.0 PL=8
MOVL C00283 V=800.0 PL=8
MOVL C00284 V=800.0 PL=8
SPYOF
MOVL C00285 V=800.0 PL=0
MOVJ C00286 VJ=25.00 PL=0
MOVL C00287 V=800.0 PL=8
SPYON
MOVL C00288 V=800.0 PL=8
MOVL C00289 V=800.0 PL=8
MOVL C00290 V=800.0 PL=8
MOVL C00291 V=800.0 PL=8
MOVL C00292 V=800.0 PL=8
MOVL C00293 V=800.0 PL=8
MOVL C00294 V=800.0 PL=8
MOVL C00295 V=800.0 PL=8
MOVL C00296 V=800.0 PL=8
MOVL C00297 V=800.0 PL=8
MOVL C00298 V=800.0 PL=8
MOVL C00299 V=800.0 PL=8
MOVL C00300 V=800.0 PL=8
MOVL C00301 V=800.0 PL=8
MOVL C00302 V=800.0 PL=8
MOVL C00303 V=800.0 PL=8
MOVL C00304 V=800.0 PL=8
MOVL C00305 V=800.0 PL=8
MOVL C00306 V=800.0 PL=8
MOVL C00307 V=800.0 PL=8
MOVL C00308 V=800.0 PL=8
MOVL C00309 V=800.0 PL=8
MOVL C00310 V=800.0 PL=8
MOVL C00311 V=800.0 PL=8
MOVL C00312 V=800.0 PL=8
MOVL C00313 V=800.0 PL=8
MOVL C00314 V=800.0 PL=8
SPYOF
MOVL C00315 V=800.0 PL=0
MOVJ C00316 VJ=25.00 PL=0
MOVL C00317 V=800.0 PL=8
SPYON
MOVL C00318 V=800.0 PL=8
MOVL C00319 V=800.0 PL=8
MOVL C00320 V=800.0 PL=8
MOVL C00321 V=800.0 PL=8
MOVL C00322 V=800.0 PL=8
MOVL C00323 V=800.0 PL=8
MOVL C00324 V=800.0 PL=8
MOVL C00325 V=800.0 PL=8
MOVL C00326 V=800.0 PL=8
MOVL C00327 V=800.0 PL=8
MOVL C00328 V=800.0 PL=8
MOVL C00329 V=800.0 PL=8
MOVL C00330 V=800.0 PL=8
MOVL C00331 V=800.0 PL=8
MOVL C00332 V=800.0 PL=8
MOVL C00333 V=800.0 PL=8
MOVL C00334 V=800.0 PL=8
MOVL C00335 V=800.0 PL=8
MOVL C00336 V=800.0 PL=8
MOVL C00337 V=800.0 PL=8
MOVL C00338 V=800.0 PL=8
MOVL C00339 V=800.0 PL=8
MOVL C00340 V=800.0 PL=8
MOVL C00341 V=800.0 PL=8
MOVL C00342 V=800.0 PL=8
MOVL C00343 V=800.0 PL=8
MOVL C00344 V=800.0 PL=8
MOVL C00345 V=800.0 PL=8
SPYOF
MOVL C00346 V=800.0 PL=0
MOVJ C00347 VJ=25.00 PL=0
MOVL C00348 V=800.0 PL=8
SPYON
MOVL C00349 V=800.0 PL=8
MOVL C00350 V=800.0 PL=8
MOVL C00351 V=800.0 PL=8
MOVL C00352 V=800.0 PL=8
MOVL C00353 V=800.0 PL=8
MOVL C00354 V=800.0 PL=8
MOVL C00355 V=800.0 PL=8
MOVL C00356 V=800.0 PL=8
MOVL C00357 V=800.0 PL=8
MOVL C00358 V=800.0 PL=8
MOVL C00359 V=800.0 PL=8
MOVL C00360 V=800.0 PL=8
MOVL C00361 V=800.0 PL=8
MOVL C00362 V=800.0 PL=8
MOVL C00363 V=800.0 PL=8
MOVL C00364 V=800.0 PL=8
MOVL C00365 V=800.0 PL=8
MOVL C00366 V=800.0 PL=8
MOVL C00367 V=800.0 PL=8
MOVL C00368 V=800.0 PL=8
MOVL C00369 V=800.0 PL=8
MOVL C00370 V=800.0 PL=8
MOVL C00371 V=800.0 PL=8
MOVL C00372 V=800.0 PL=8
MOVL C00373 V=800.0 PL=8
MOVL C00374 V=800.0 PL=8
MOVL C00375 V=800.0 PL=8
MOVL C00376 V=800.0 PL=8
SPYOF
MOVL C00377 V=800.0 PL=0
MOVJ C00378 VJ=25.00 PL=0
MOVL C00379 V=800.0 PL=8
SPYON
MOVL C00380 V=800.0 PL=8
MOVL C00381 V=800.0 PL=8
MOVL C00382 V=800.0 PL=8
MOVL C00383 V=800.0 PL=8
MOVL C00384 V=800.0 PL=8
MOVL C00385 V=800.0 PL=8
MOVL C00386 V=800.0 PL=8
MOVL C00387 V=800.0 PL=8
MOVL C00388 V=800.0 PL=8
MOVL C00389 V=800.0 PL=8
MOVL C00390 V=800.0 PL=8
MOVL C00391 V=800.0 PL=8
MOVL C00392 V=800.0 PL=8
MOVL C00393 V=800.0 PL=8
MOVL C00394 V=800.0 PL=8
MOVL C00395 V=800.0 PL=8
MOVL C00396 V=800.0 PL=8
MOVL C00397 V=800.0 PL=8
MOVL C00398 V=800.0 PL=8
MOVL C00399 V=800.0 PL=8
MOVL C00400 V=800.0 PL=8
MOVL C00401 V=800.0 PL=8
MOVL C00402 V=800.0 PL=8
MOVL C00403 V=800.0 PL=8
MOVL C00404 V=800.0 PL=8
MOVL C00405 V=800.0 PL=8
MOVL C00406 V=800.0 PL=8
MOVL C00407 V=800.0 PL=8
MOVL C00408 V=800.0 PL=8
MOVL C00409 V=800.0 PL=8
SPYOF
MOVL C00410 V=800.0 PL=0
MOVJ C00411 VJ=25.00 PL=0
MOVL C00412 V=800.0 PL=8
SPYON
MOVL C00413 V=800.0 PL=8
MOVL C00414 V=800.0 PL=8
MOVL C00415 V=800.0 PL=8
MOVL C00416 V=800.0 PL=8
MOVL C00417 V=800.0 PL=8
MOVL C00418 V=800.0 PL=8
MOVL C00419 V=800.0 PL=8
MOVL C00420 V=800.0 PL=8
MOVL C00421 V=800.0 PL=8
MOVL C00422 V=800.0 PL=8
MOVL C00423 V=800.0 PL=8
MOVL C00424 V=800.0 PL=8
MOVL C00425 V=800.0 PL=8
MOVL C00426 V=800.0 PL=8
MOVL C00427 V=800.0 PL=8
MOVL C00428 V=800.0 PL=8
MOVL C00429 V=800.0 PL=8
MOVL C00430 V=800.0 PL=8
MOVL C00431 V=800.0 PL=8
MOVL C00432 V=800.0 PL=8
MOVL C00433 V=800.0 PL=8
MOVL C00434 V=800.0 PL=8
MOVL C00435 V=800.0 PL=8
MOVL C00436 V=800.0 PL=8
MOVL C00437 V=800.0 PL=8
SPYOF
MOVL C00438 V=800.0 PL=0
MOVJ C00439 VJ=25.00 PL=0
MOVL C00440 V=800.0 PL=8
SPYON
MOVL C00441 V=800.0 PL=8
MOVL C00442 V=800.0 PL=8
MOVL C00443 V=800.0 PL=8
MOVL C00444 V=800.0 PL=8
MOVL C00445 V=800.0 PL=8
MOVL C00446 V=800.0 PL=8
MOVL C00447 V=800.0 PL=8
MOVL C00448 V=800.0 PL=8
MOVL C00449 V=800.0 PL=8
MOVL C00450 V=800.0 PL=8
MOVL C00451 V=800.0 PL=8
SPYOF
MOVL C00452 V=800.0 PL=8
MOVJ C00453 VJ=25.00 PL=8
MOVL C00454 V=800.0 PL=8
MOVL C00455 V=800.0 PL=8
MOVJ C00456 VJ=25.00 PL=8
MOVL C00457 V=800.0 PL=8
SPYON
MOVL C00458 V=800.0 PL=8
SPYOF
MOVL C00459 V=800.0 PL=8
MOVJ C00460 VJ=25.00 PL=8
MOVL C00461 V=800.0 PL=8
SPYON
MOVL C00462 V=800.0 PL=8
SPYOF
MOVL C00463 V=800.0 PL=8
MOVJ C00464 VJ=25.00 PL=8
'Path End
MOVJ C00465 VJ=100.00 PL=8
END
